FUNCTION_BLOCK Stage10 (* Template for a Basic Function Block Type *)
  (* Standard: 61499-2 *)
  (* Version 1.0, 2021-06-20, HP *)
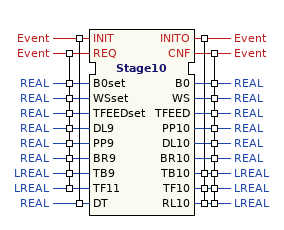
  EVENT_INPUT
    INIT WITH DT; (* Initialization Request *)
    REQ WITH B0set, WSset, TFEEDset, DL9, PP9, BR9, TB9, TF11; (* Normal Execution Request *)
  END_EVENT
  EVENT_OUTPUT
    INITO WITH RL10, TF10, TB10; (* Initialization Confirm *)
    CNF WITH PP10, TFEED, B0, WS, DL10, BR10, TB10, TF10, RL10; (* Execution Confirmation *)
  END_EVENT
  VAR_INPUT
    B0set : REAL;
    WSset : REAL;
    TFEEDset : REAL;
    DL9 : REAL;
    PP9 : REAL;
    BR9 : REAL;
    TB9 : LREAL;
    TF11 : LREAL;
    DT : REAL;
  END_VAR
  VAR_OUTPUT
    B0 : REAL;
    WS : REAL;
    TFEED : REAL;
    PP10 : REAL;
    DL10 : REAL;
    BR10 : REAL;
    TB10 : LREAL;
    TF10 : LREAL;
    RL10 : LREAL;
  END_VAR
  VAR
    AB : REAL; (* internal variabel *)
    UU : REAL;
    TREF : REAL;
    AD : REAL;
    AHC : REAL;
    AHR : REAL;
    AS : REAL;
    REC : REAL;
    WN : REAL;
    WN_1 : REAL;
    XKN : REAL;
    C1 : REAL;
    HS : REAL;
    G : REAL;
    W1 : REAL;
    TFREC : REAL;
    TS : REAL;
    DTS : REAL;
    TF10_last : REAL;
    RL10_last : REAL;
    TB10_last : REAL;
    USS : REAL;
    RHOB : REAL;
    CPB : REAL;
    CPF : REAL;
    FMW : REAL;
    HLV : REAL;
    HV : REAL;
    BPR : REAL;
    FMC : REAL;
    U : REAL;
    A : REAL;
    B : REAL;
    C : REAL;
    D1 : REAL;
    d : REAL;
    a : REAL;
    A1 : REAL;
    A2 : REAL;
    A3 : REAL;
    A4 : REAL;
    A5 : REAL;
    A6 : REAL;
    p : REAL;
    q : REAL;
    TC : REAL;
    PC : REAL;
    DTB10 : REAL;
    DEN10 : REAL;
    DH10 : REAL;
    DP10 : REAL;
    DPDH10 : REAL;
    DT10 : REAL;
    m : REAL;
    n : REAL;
    VR10 : REAL;
    DELTA10 : REAL;
    DELTA32 : REAL;
    DELTA54 : REAL;
    DELTA10_last : REAL;
    DELTA32_last : REAL;
    DELTA54_last : REAL;
  END_VAR
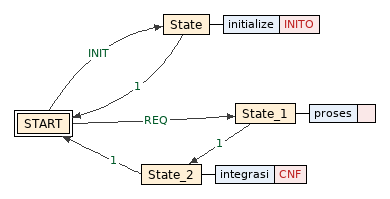
  EC_STATES
    START; (* Initial State *)
    State : initialize -> INITO;
    State_1 : proses;
    State_2 : integrasi -> CNF;
  END_STATES
  EC_TRANSITIONS
    START TO State := INIT;
    State TO START := 1;
    START TO State_1 := REQ;
    State_1 TO State_2 := 1;
    State_2 TO START := 1;
  END_TRANSITIONS
  ALGORITHM initialize IN ST: (* Initialization algorithm *)
TREF :=273.15;
AB :=57.2727;
AHC :=4069.2;
AHR :=2639.7;
AS :=3225.7;
REC :=0.0;
//TF2:=TF2;

//TFEED :=TFEED1+TREF;
 //TS:=TS1+TREF;
WN :=3.0;
XKN :=0.68;
HS:=0.11;
G :=9.81;
W1 :=0.50;

RL10 := 0.572892175112335;
TB10 := 340.514997951413;
TF10 := 336.687818219045;
TF11 := 334.143160422222;


RL10_last :=RL10;
TB10_last :=TB10;
TF10_last :=TF10;
  END_ALGORITHM
  ALGORITHM proses IN ST: (* kalkulasi *)
B0 :=B0set;
WS :=WSset;
TFEED:=TFEEDset;
UU := TFEEDset;
U :=UU;

USS :=49.767;
C1 :=0.625;
RHOB :=1032.4; //maassa jenis brine
CPB :=1.00; //heatcapacity Brine
CPF :=1.00; //heat capacity feed
FMW :=23654.0;
HLV :=563.7959;
HV :=625.1971;
BPR :=2.192;
FMC :=34736.09;
//U :=UU; //feed temp



///  Calculate the physical properties

//A :=3.2437814;
//B :=5.86826*0.001;
//C :=1.1702379*0.00000001;
//D1 :=2.1878462*0.001;
//TC :=647.27;
//PC :=218.167;


A1 :=3.2437814;
A2:=5.86826*0.001;
A3:=1.1702379*0.00000001;
A4 :=2.1878462*0.001;
A5 :=647.27;
A6 :=218.167;

DTB10 :=A5-TB10;
DEN10 :=(A1+A2*DTB10+A3*DTB10*DTB10*DTB10)/(1+A4*DTB10)*DTB10/TB10;
p:=DEN10;
q:=10.0;
PP10 :=A6/(EXPT(q, p));

// calculate the brine flow rates
DP10:=PP9-PP10;
DH10:=RL10-C1*HS;
DPDH10 :=DP10*101000+G*RHOB*DH10;
m:=DPDH10*RHOB;
n:=0.5;
BR10 :=WN*XKN*RL10*(EXPT(m, n));
BR10 :=BR10*60.0/1000.0;

// calculate the vapor flow rates

DT10 :=TB10-BPR/1.8-(TF11+TF10)*0.5;
VR10:=U*AHC*DT10/HLV/1000.0;
DL10 :=DL9+VR10;


//// state equation
DELTA10 :=(BR9-BR10-VR10)*1000.0/RHOB/AB;
DELTA32 :=((BR9*CPB*(TB9-TB10))-VR10*(HV-CPB*(TB10-TREF)))*1000.0/AB/RHOB/CPB/RL10;
DELTA54 :=(B0*CPF*(TF11-TF10)*1000+(U*AHC*DT10))/FMW/CPF;
  END_ALGORITHM
  ALGORITHM integrasi IN ST: (* new algorithm *)
B0 :=B0set;
WS :=WSset;
TFEED:=TFEEDset;
//integrasi
RL10 := (DELTA10 + DELTA10_last)*0.5*DT + RL10_last;
DELTA10_last :=DELTA10 ;
RL10_last :=RL10;

TB10:= (DELTA32 + DELTA32_last)*0.5*DT + TB10_last;
DELTA32_last :=DELTA32 ;
TB10_last:=TB10;

TF10 := (DELTA54 + DELTA54_last)*0.5*DT + TF10_last;
DELTA54_last :=DELTA54 ;
TF10_last :=TF10;
  END_ALGORITHM
END_FUNCTION_BLOCK
